// TIA Portal V19 export
TYPE "C501_VAR_BWR_TYPIC"
   STRUCT
      BSC { ExternalAccessible := 'False'; ExternalVisible := 'False'; ExternalWritable := 'False'} : USInt;   // Beschikbaarheidsstatus
   END_STRUCT;
END_TYPE
